{attribute 'TcGenerated'}
// This function has been automatically generated from the project information.
VAR_GLOBAL CONSTANT
    {attribute 'const_non_replaced'}
    {attribute 'linkalways'}
    stLibVersion_lcls_plc_xrt_optics : ST_LibVersion := (iMajor := 3, iMinor := 1, iBuild := 0, iRevision := 0, sVersion := '3.1.0');
END_VAR

(* stored: Version 1.1.0.1, ProductVersion 3.1.4020.12
   GVL Global_Version: Id 3a5b10c6-bfaf-4fb7-b8d1-512005083c0d *)
